// TwinCAT 3 PLC project FunctionBlocks
// ProgramVersion: 3.1.4023.0
// libraries:
//   Tc2_ControllerToolbox, * (Beckhoff Automation GmbH)
//   Tc2_Standard, * (Beckhoff Automation GmbH)
//   Tc2_System, * (Beckhoff Automation GmbH)
//   Tc3_Module, * (Beckhoff Automation GmbH)
// project tree:
//   DUTs/ dut_Auto_rock.TcDUT, dut_Brake.TcDUT, dut_Clutch.TcDUT, dut_Dol_Starter.TcDUT, ST_CSV_Record.TcDUT (not stored), S_Drive_control_settings.TcDUT, dut_hmi_Analogue.TcDUT, dut_hmi_Depth.TcDUT, dut_hmi_Drive_control.TcDUT, dut_hmi_Power_lever.TcDUT, dut_Least_gate.TcDUT, dut_Mode.TcDUT, dut_Power_lever.TcDUT, dut_Safety.TcDUT, S_TPD32_base_settings.TcDUT, S_General_settings.TcDUT
//   GVLs/ Brakes.TcGVL, Clutch.TcGVL, GVL.TcGVL, Mode.TcGVL, Power_lever.TcGVL, Safety.TcGVL, sp.TcGVL, Torque_prediction.TcGVL
//   / PlcTask.TcTTO
//   POUs/FBs/ FB_Brake_oil_pump.TcPOU, FB_Ctl_cmd_u.TcPOU, FB_DOL_Control.TcPOU, FB_Escort_monitoring.TcPOU, FB_Analogue.TcPOU, FB_Analogue_xcheck.TcPOU, FB_Auto_rock.TcPOU, FB_Backout.TcPOU, FB_BIT_TO_WORD_V0.TcPOU, FB_Brake.TcPOU, FB_Clutch.TcPOU, FB_Disc_brake.TcPOU, FB_Double_drum.TcPOU, FB_Drive_control.TcPOU, FB_Duty.TcPOU, FB_Encoder_depth.TcPOU, FB_Fast_brake.TcPOU, FB_Hysteresis.TcPOU, FB_Lag_filter.TcPOU, FB_Least_gate_element.TcPOU, FB_Least_gate_result.TcPOU, FB_Lincon.TcPOU, FB_Mode.TcPOU, FB_Motor_run_time.TcPOU, FB_Moving_average.TcPOU, FB_No_start.TcPOU, FB_Power_lever.TcPOU, FB_Raw_to_scaled.TcPOU, FB_Ref_ramp.TcPOU, FB_sp_write.TcPOU (not stored), FB_Standard_stuff.TcPOU, FB_Torque_prediction.TcPOU, FB_Torque_prediction_ST.TcPOU, FB_TPD_CANopen.TcPOU, FB_TP_with_stop.TcPOU, FB_Trip_control.TcPOU, FB_Valve_monitor.TcPOU, FB_Window.TcPOU, FB_WORD_TO_BIT_V0.TcPOU
//   POUs/ MAIN.TcPOU
//   POUs/Sections/ Winder_data.TcPOU
// real-time tasks:
//   TASK PlcTask: cycle T#10ms, priority 20, ADS port 350

CONFIGURATION FunctionBlocks
    RESOURCE PLC ON TwinCAT3
        TASK PlcTask(INTERVAL := T#10ms, PRIORITY := 20);
        PROGRAM MAIN WITH PlcTask : MAIN;
    END_RESOURCE
END_CONFIGURATION

// ---- DUTs/dut_Auto_rock.TcDUT
TYPE dut_Auto_rock :
STRUCT
	Status:WORD;
	Command:WORD;
END_STRUCT
END_TYPE

// ---- DUTs/dut_Brake.TcDUT
TYPE dut_Brake :
STRUCT
	Lh_off:BOOL;(*Left brake off signal - usually from left spring nest*)
	Lh_rubbing:BOOL; (*Left brake rubbing signal - usually from left spring nest*)
	Lh_on:BOOL; (*Left brake on signal - usually from left spring nest*)
	Lh_wear:BOOL; (*Left brake wear signal - usually from left spring nest*)
	Rh_off:BOOL; (*Right brake on signal - usually from right spring nest*)
	Rh_rubbing:BOOL; (*Right brake rubbing signal - usually from right spring nest*)
	Rh_on:BOOL; (*Right brake on signal - usually from right spring nest*)
	Rh_wear:BOOL; (*Right brake wear signal - usually from Right spring nest*)
	Lever_on:BOOL; (*Brake lever on limit switch*)
	Lever_off:BOOL; (*Brake lever off - normally from same limit switch as 'Lever_on'*)
	Lever_fully_off:BOOL; (*Brake lever fully off limit switch. Necessary for automatic winders.*)
	Maintenance_switch:BOOL; (*Brake maintenance switch (can be on driver's desk or in control panels).*)
	Maintenance_mode:BOOL;
	Lh_test:BOOL; (*Left brake test switch - normally on driver's desk. Often the same switch as Lh_dump.*)
	Rh_test:BOOL; (*Right brake test switch - normally on driver's desk. Often the same switch as Rh_dump.*)
	Lh_dump:BOOL; (*Left brake dump switch - normally on driver's desk. Often the same switch as Lh_test.*)
	Rh_dump:BOOL; (*Right brake dump switch - normally on driver's desk. Often the same switch as Rh_test.*)
	Proved_on:BOOL;
	Proved_on_500ms:BOOL;
END_STRUCT
END_TYPE

// ---- DUTs/dut_Clutch.TcDUT
TYPE dut_Clutch :
STRUCT
	Lh_in:BOOL;
	Lh_out:BOOL;
	Rh_in:BOOL;
	Rh_out:BOOL;
	Single_drum:BOOL;
END_STRUCT
END_TYPE

// ---- DUTs/dut_Dol_Starter.TcDUT
TYPE dut_Dol_Starter :
STRUCT
	Input_word:WORD; (*0=Switch, 1=Run, 2=Trip, 3=NoStart, 4=Estop, 5=IL1, 6=IL2, 7=IL3*)
	Output_word:WORD;
	Hrs:REAL;
	Minutes:REAL;
	Sec:REAL;
END_STRUCT
END_TYPE

// ---- DUTs/S_Drive_control_settings.TcDUT
TYPE S_Drive_control_settings :
STRUCT
	Max_drive_speed:INT;
	Max_drive_torque:INT;
	Speed_S_func_scans:INT;
	Current_S_func_scans:INT;
	No_start_time:TIME;
	Motor_fed_delay:TIME;
	Stall_time:TIME;
	Stall_speed:INT;
	Torque_ctrl_max_speed:INT;
	Brake_apply_speed:INT;
	Trail_brake_speed:INT;
	De_energise_to_trail:BOOL;
	Single_lever_control:BOOL;
	Stall_current:INT;
	Backout_min_speed:INT;

	(*Torque prediction settings*)	
	Lh_cage_mass_current:REAL;
	Rh_cage_mass_current:REAL;
	Lh_rope_mass_current:REAL;
	Rh_rope_mass_current:REAL;
	Full_payload_current:REAL;
	A_s2_per_m:REAL;
	Accel_torque_lag:TIME;
	Dynamic_friction_current:REAL;

END_STRUCT
END_TYPE

// ---- DUTs/dut_hmi_Analogue.TcDUT
TYPE dut_hmi_Analogue :
STRUCT
	Value:REAL;
	Per_thousand:REAL;
	Colour:INT;
END_STRUCT
END_TYPE

// ---- DUTs/dut_hmi_Depth.TcDUT
TYPE dut_hmi_Depth :
STRUCT
	Raw_count:REAL;
	Corrected_count:REAL;
	Raw_depth:REAL;
	Calibrated_depth:REAL;
	Compensated_depth:REAL;
	Offset:REAL;
	Speed:REAL;
	Status:WORD;
END_STRUCT
END_TYPE

// ---- DUTs/dut_hmi_Drive_control.TcDUT
TYPE dut_hmi_Drive_control :
STRUCT
	Speed_ref:INT;
	Torque_ref:INT;
	Torque_prediction:INT;
	Speed_scale:INT;
	Driver_ref_final:INT;
	Status:WORD;
END_STRUCT
END_TYPE

// ---- DUTs/dut_hmi_Power_lever.TcDUT
TYPE dut_hmi_Power_lever :
STRUCT
	Status:WORD;
	Raw:INT;
	Linear:INT;
	Cubic:INT;
END_STRUCT
END_TYPE

// ---- DUTs/dut_Least_gate.TcDUT
TYPE dut_Least_gate :
STRUCT
	Min_allowed_speed:REAL;
	Description:STRING[16];
	Rope_cap_mode:BOOL;
END_STRUCT
END_TYPE

// ---- DUTs/dut_Mode.TcDUT
TYPE dut_Mode :
STRUCT
	Manual:BOOL;
	Auto:BOOL;
	Auto_go:BOOL;
	Men:BOOL;
	Material:BOOL;
	Rope_capping:BOOL;
	Brake_maintenance:BOOL;
	Manual_switch:BOOL;
	Auto_switch:BOOL;
	Men_switch:BOOL;
	Material_switch:BOOL;
	Rope_capping_switch:BOOL;
	Rock:BOOL;
	Single_lever_control:BOOL;
END_STRUCT
END_TYPE

// ---- DUTs/dut_Power_lever.TcDUT
TYPE dut_Power_lever :
STRUCT
	Neutral:BOOL;
	Forward:BOOL;
	Reverse:BOOL;
	Button:BOOL;
	Raw:INT;
	Linear:INT;
	Cubic:INT;
END_STRUCT
END_TYPE

// ---- DUTs/dut_Safety.TcDUT
TYPE dut_Safety :
STRUCT
	Sc1:BOOL;
	Sc2:BOOL;
	Busc1:BOOL;
	Busc2:BOOL;
	Backup_safety_trip:BOOL;
	Main_safety_trip:BOOL;
	Lily_func_trip:BOOL;
	Lily_app_fault:BOOL;
	Backup_control_trip:BOOL;
	Control_trip:BOOL;
	Control_stop:BOOL;
	Lockout:BOOL;
	Enforced_slow:BOOL;
	Alarm:BOOL;
	All_clear:BOOL;
	Reset_button:BOOL;
	Reset_interlocks:BOOL;
	Reset:BOOL;
	Safe_for_power:BOOL;
	Bridge_present:BOOL;
END_STRUCT
END_TYPE

// ---- DUTs/S_TPD32_base_settings.TcDUT
TYPE S_TPD32_base_settings :
STRUCT
	Motor_base_rpm:REAL; (*Rated rpm of the motor*)
	Max_output_voltage:REAL; (*Maximum DC armature voltage*)
	Full_load_curr:REAL; (*Rated armature amps of the motor*)
	DCV_nominal_flux_current:REAL; (*Nominal flux current of the DCV according to S14 DIP switches*)
	Motor_nominal_flux_current:REAL; (*Nominal flux current of the DCV according to S14 DIP switches*)
	Flux_current_min:REAL; (*Percentage of rated motor field current for field weakening*)
	Acc_delta_time:REAL; (*Acceleration time from zero to rated motor rpm in seconds*)
	Dec_delta_time:REAL; (*Deceleration time from rated motor rpm to zero in seconds*)
END_STRUCT
END_TYPE

// ---- DUTs/S_General_settings.TcDUT
TYPE S_General_settings :
STRUCT
	Full_speed: REAL;
	Slow_switch_speed: REAL;
END_STRUCT
END_TYPE

// ---- GVLs/Brakes.TcGVL
{attribute 'qualified_only'}
VAR_GLOBAL
	Lh_off:BOOL;(*Left brake off signal - usually from left spring nest*)
	Lh_rubbing:BOOL; (*Left brake rubbing signal - usually from left spring nest*)
	Lh_on:BOOL; (*Left brake on signal - usually from left spring nest*)
	Lh_wear:BOOL; (*Left brake wear signal - usually from left spring nest*)
	Rh_off:BOOL; (*Right brake on signal - usually from right spring nest*)
	Rh_rubbing:BOOL; (*Right brake rubbing signal - usually from right spring nest*)
	Rh_on:BOOL; (*Right brake on signal - usually from right spring nest*)
	Rh_wear:BOOL; (*Right brake wear signal - usually from Right spring nest*)
	Lever_on:BOOL; (*Brake lever on limit switch*)
	Lever_off:BOOL; (*Brake lever off - normally from same limit switch as "Lever_on"*)
	Lever_fully_off:BOOL; (*Brake lever fully off limit switch. Necessary for automatic winders.*)
	Maintenance_switch:BOOL; (*Brake maintenance switch (can be on driver's desk or in control panels).*)
	Maintenance_mode:BOOL;
	Lh_test:BOOL; (*Left brake test switch - normally on driver's desk. Often the same switch as Lh_dump.*)
	Rh_test:BOOL; (*Right brake test switch - normally on driver's desk. Often the same switch as Rh_dump.*)
	Lh_dump:BOOL; (*Left brake dump switch - normally on driver's desk. Often the same switch as Lh_test.*)
	Rh_dump:BOOL; (*Right brake dump switch - normally on driver's desk. Often the same switch as Rh_test.*)
	Proved_on:BOOL;
	Proved_on_500ms:BOOL;
END_VAR

// ---- GVLs/Clutch.TcGVL
{attribute 'qualified_only'}
VAR_GLOBAL
	Lh_in:BOOL;
	Lh_out:BOOL;
	Rh_in:BOOL;
	Rh_out:BOOL;
	Single_drum:BOOL;
END_VAR

// ---- GVLs/GVL.TcGVL
{attribute 'qualified_only'}
VAR_GLOBAL
	Mode:dut_Mode;
	Brakes:dut_Brake;
	Clutch:dut_Clutch;
	Power_lever:dut_Power_lever;
	Safety:dut_Safety;
END_VAR

// ---- GVLs/Mode.TcGVL
{attribute 'qualified_only'}
VAR_GLOBAL
	Manual:BOOL;
	Auto:BOOL;
	Auto_go:BOOL;
	Men:BOOL;
	Material:BOOL;
	Rope_capping:BOOL;
	Brake_maintenance:BOOL;
	Manual_switch:BOOL;
	Auto_switch:BOOL;
	Men_switch:BOOL;
	Material_switch:BOOL;
	Rope_capping_switch:BOOL;
	Rock:BOOL;
	Single_lever_control:BOOL;
END_VAR

// ---- GVLs/Power_lever.TcGVL
{attribute 'qualified_only'}
VAR_GLOBAL
	Neutral:BOOL;
	Forward:BOOL;
	Reverse:BOOL;
	Button:BOOL;
	Raw:INT;
	Linear:INT;
	Cubic:INT;
END_VAR

// ---- GVLs/Safety.TcGVL
{attribute 'qualified_only'}
VAR_GLOBAL
	Sc1:BOOL;
	Sc2:BOOL;
	Busc1:BOOL;
	Busc2:BOOL;
	Backup_safety_trip:BOOL;
	Main_safety_trip:BOOL;
	Lily_func_trip:BOOL;
	Lily_app_fault:BOOL;
	Backup_control_trip:BOOL;
	Control_trip:BOOL;
	Control_stop:BOOL;
	Lockout:BOOL;
	Enforced_slow:BOOL;
	Alarm:BOOL;
	All_clear:BOOL;
	Reset_button:BOOL;
	Reset_interlocks:BOOL;
	Reset:BOOL;
	Safe_for_power:BOOL;
	Bridge_present:BOOL;
END_VAR

// ---- GVLs/sp.TcGVL
{attribute 'qualified_only'}
VAR_GLOBAL
	Gen: S_General_settings;
	Drive: S_Drive_control_settings;
	TPD: S_TPD32_base_settings;
END_VAR

// ---- GVLs/Torque_prediction.TcGVL
{attribute 'qualified_only'}
VAR_GLOBAL
	Lh_full: BOOL;
	Lh_half: BOOL;
	Equal: BOOL;
	Rh_half: BOOL;
	Rh_full: BOOL;
	
	Lh_full_request: BOOL;
	Lh_half_request: BOOL;
	Equal_request: BOOL;
	Rh_half_request: BOOL;
	Rh_full_request: BOOL;
END_VAR

// ---- POUs/MAIN.TcPOU
PROGRAM MAIN
VAR
END_VAR

END_PROGRAM

// ---- POUs/FBs/FB_Brake_oil_pump.TcPOU
FUNCTION_BLOCK FB_Brake_oil_pump
VAR_INPUT
	Run_cmd:BOOL;
	Stop_cmd:BOOL;
	Bop1_switch:BOOL;
	Bop1_tripped:BOOL;
	Bop1_running:BOOL;
	Bop1_use_internal_es:BOOL;
	Bop1_ext_estop:BOOL;
	Bop2_switch:BOOL;
	Bop2_tripped:BOOL;
	Bop2_running:BOOL;
	Bop2_use_internal_es:BOOL;
	Bop2_ext_estop:BOOL;
	Bop1_interlock:BOOL;
	Bop2_interlock:BOOL;
	Common_interlock:BOOL;
	Bridge1:BOOL;
	Bridge2:BOOL;
	Bridge3:BOOL;
	Pause_time:TIME;
	Reset:BOOL;
	Duty_bop1:REAL;
	Duty_bop2:REAL;
	Bop1_Reg455:REAL;
	Bop2_Reg455:REAL;
END_VAR
VAR_OUTPUT
	Bop1_run:BOOL;
	Bop2_run:BOOL;
	Bop1_ns_trip:BOOL;
	Bop1_es_trip:BOOL;
	Bop1_contactor_stuck:BOOL;
	Bop2_ns_trip:BOOL;
	Bop2_es_trip:BOOL;
	Bop2_contactor_stuck:BOOL;
	Start_output:BOOL;
	Bop1_Reg704:REAL;
	Bop1_Reg703:REAL;
	Bop1_Avg_curr:REAL;
	Bop2_Reg704:REAL;
	Bop2_Reg703:REAL;
	Bop2_Avg_curr:REAL;
END_VAR
VAR_IN_OUT
	Bop1_data:dut_Dol_Starter;
	Bop2_data:dut_Dol_Starter;
END_VAR
VAR
	FB_Duty_0: FB_Duty;
	FB_DOL_Control_0: FB_DOL_Control;
	FB_DOL_Control_1: FB_DOL_Control;
END_VAR

M_Brake_oil_pump();

METHOD M_Brake_oil_pump
VAR_INPUT
END_VAR
VAR_INST // added by the converter: edge detectors and wires of the graphical bodies
    _w1 : BOOL;
END_VAR
Start_output := _w1;
Bop1_avg_curr := FB_DOL_Control_0.Avg_curr;
Bop2_run := FB_DOL_Control_1.Fwd_command;
Bop1_run := FB_DOL_Control_0.Fwd_command;
Bop2_ns_trip := FB_DOL_Control_1.Ns_trip;
Bop2_es_trip := FB_DOL_Control_1.Estop_trip;
Bop2_contactor_stuck := FB_DOL_Control_1.Contactor_stuck;
Bop2_Reg704 := FB_DOL_Control_1.Reg_704;
Bop2_Reg703 := FB_DOL_Control_1.Reg_703;
_w1 := FB_DOL_Control_0.Start_output OR FB_DOL_Control_1.Start_output;
Bop1_ns_trip := FB_DOL_Control_0.Ns_trip;
Bop1_es_trip := FB_DOL_Control_0.Estop_trip;
Bop1_contactor_stuck := FB_DOL_Control_0.Contactor_stuck;
Bop1_Reg704 := FB_DOL_Control_0.Reg_704;
Bop2_avg_curr := FB_DOL_Control_1.Avg_curr;
Bop1_Reg703 := FB_DOL_Control_0.Reg_703;
FB_DOL_Control_1(
    Run_fwd := Run_cmd,
    Stop := Stop_cmd,
    Breaker_on := Bop2_switch,
    Breaker_tripped := Bop2_tripped,
    Contactor_feedback := Bop2_running,
    Interlock2 := Bop2_interlock,
    Bridge2 := Bridge2,
    Interlock3 := Common_interlock,
    Bridge3 := Bridge3,
    Reset := Reset,
    Use_internal_ES := Bop2_use_internal_es,
    Ext_estop := Bop2_ext_estop,
    Pause_time := Pause_time,
    Duty := FB_Duty_0.DutyB,
    Reg_455 := Bop2_Reg455,
    Starter_data := Bop2_data); // FB_DOL_Control
FB_DOL_Control_0(
    Run_fwd := Run_cmd,
    Stop := Stop_cmd,
    Breaker_on := Bop1_switch,
    Breaker_tripped := Bop1_tripped,
    Contactor_feedback := Bop1_running,
    Interlock1 := Bop1_interlock,
    Bridge1 := Bridge1,
    Interlock3 := Common_interlock,
    Bridge3 := Bridge3,
    Reset := Reset,
    Use_internal_ES := Bop1_use_internal_es,
    Ext_estop := Bop1_ext_estop,
    Pause_time := Pause_time,
    Duty := FB_Duty_0.DutyA,
    Reg_455 := Bop1_Reg455,
    Starter_data := Bop1_data); // FB_DOL_Control
FB_Duty_0(
    DutyA_times := Duty_bop1,
    DeviceA_running := Bop1_data.Input_word.1,
    DeviceA_switch := Bop1_data.Input_word.0,
    Force_dutyA := Bop1_data.Input_word.5,
    DutyB_times := Duty_bop2,
    Device_B_running := Bop2_data.Input_word.1,
    DeviceB_switch := Bop2_data.Input_word.0,
    Force_dutyB := Bop2_data.Input_word.5); // FB_Duty
END_METHOD

END_FUNCTION_BLOCK

// ---- POUs/FBs/FB_Duty.TcPOU
FUNCTION_BLOCK FB_Duty
VAR_INPUT
	DutyA_times:REAL; (*Times that Device A must run*)
	DeviceA_running:BOOL; (*Device A contactor feedback(running signal)*)
	DeviceA_switch:BOOL;
	DeviceA_ns:BOOL; (*Device A No Start - Switch duty to B*)
	Force_dutyA:BOOL;
	DutyB_times:REAL; (*Time that Device B must run*)
	DeviceB_running:BOOL; (*Device B contactor feedback(running signal)*)
	DeviceB_switch:BOOL;
	DeviceB_ns:BOOL; (*Device B No Start - Switch duty to A*)
	Force_dutyB:BOOL;
END_VAR
VAR_OUTPUT
	DutyA:BOOL; (*Device A output*)
	DutyB:BOOL; (*Device B output*)
END_VAR
VAR
	DeviceA_runtime:REAL;
	DeviceA_running_GT_1s:BOOL;
	DA_runtime:TIME;
	DeviceB_runtime:REAL;
	DeviceB_running_GT_1s:BOOL;
	DB_runtime:TIME;
	FE_bit_A :BOOL;
	FE_bit_B :BOOL;
	F_TRIG_0: F_TRIG;
	F_TRIG_1: F_TRIG;
	TON_2 : TON;
	TON_3 : TON;
END_VAR

M_Duty();

METHOD M_Duty
VAR_INPUT
END_VAR
IF NOT DeviceA_switch THEN
	DeviceA_runtime :=0;
end_if;
 
if NOT DeviceB_switch then
	DeviceB_runtime :=0;
end_if;

if NOT Force_dutyA and NOT Force_dutyB then
	if DeviceA_switch then
		IF DeviceA_runtime < DutyA_times AND NOT DutyB THEN
			DutyA := True;
		END_IF;
		F_TRIG_0(CLK:= DeviceA_running_GT_1s, Q=> FE_bit_A);
		IF FE_bit_A THEN
			DeviceA_runtime := DeviceA_runtime +1;
		end_if;
		if DeviceA_runtime >= DutyA_times and NOT Force_dutyA then
			DutyA := False;
			DeviceA_runtime := 0;
		end_if;

	end_if;


	if DeviceB_switch then
		IF DeviceB_runtime < DutyB_times AND NOT DutyA THEN
			DutyB := True;
		END_IF;
		F_TRIG_1(CLK:= DeviceB_running_GT_1s, Q=> FE_bit_B);
		IF FE_bit_B THEN
			DeviceB_runtime := DeviceB_runtime +1;
		end_if;
		if DeviceB_runtime >= DutyB_times and NOT Force_dutyB then
			DutyB := False;
			DeviceB_runtime := 0;
		end_if;
	end_if;

end_if;

if (Force_dutyA and DeviceA_switch) or (DeviceA_switch and NOT DeviceB_switch)  then
	DutyA := True;
	DutyB := False;
	DeviceA_runtime := 0;
	DeviceB_runtime := 0;
end_if;

if Force_dutyB and DeviceB_switch  or (DeviceB_switch and NOT DeviceA_switch) then
	DutyB := True;
	DutyA := False;
	DeviceA_runtime := 0;
	DeviceB_runtime := 0;
END_IF;

TON_2 (IN := DeviceA_running,
       PT := t#2s,
       Q => DeviceA_running_GT_1s,
       ET => DA_runtime);

TON_3 (IN := DeviceB_running,
       PT := t#2s,
       Q => DeviceB_running_GT_1s,
       ET => DB_runtime);
END_METHOD

END_FUNCTION_BLOCK

// ---- POUs/FBs/FB_DOL_Control.TcPOU
FUNCTION_BLOCK FB_DOL_Control
VAR_INPUT
	Run_fwd:BOOL; (*Pulsed Input to run forward*)
	Run_rev:BOOL; (*Pulsed Input to run reverse*)
	Stop:BOOL; (*Stop command*)
	Breaker_on:BOOL; (*Circuit breaker On status*)
	Breaker_tripped:BOOL;(*Overload tripped*)
	Contactor_feedback:BOOL; (*Running Feedback*)
	Interlock1:BOOL; (*Interlock to inhibit starter output*)
	Bridge1:BOOL; (*Bridge interlock1*)
	Interlock2:BOOL; (*Interlock to inhibit starter output*)
	Bridge2:BOOL; (*Bridge interlock2*)
	Interlock3:BOOL; (*Interlock to inhibit starter output*)
	Bridge3:BOOL; (*Bridge interlock3*)
	Reset:BOOL;
	Use_internal_ES:BOOL; (*1= Use EStop , 0= Dont use*)
	Ext_estop:BOOL; (*External Monitored Estop contact*)
	Pause_time:TIME; (*Time before starting next starter*)
	Duty:BOOL; (*1= active duty*)
	Hide_duty_indication:BOOL; (*1=Hide label on HMI*)
	Reg_455:REAL;
END_VAR
VAR_OUTPUT
	Fwd_command:BOOL; (*Run forward command*)
	Rev_command:BOOL; (*Run reverse command*)
	Ns_trip:BOOL;
	Estop_trip:BOOL; (*E-Stop/ Contactor feedback loss*)
	Contactor_stuck:BOOL; (*No run command but contactor closed*)
	Tripped_out:BOOL;
	Start_output:BOOL; (*Start command to next starter block*)
	Reg_704:REAL;
	Reg_703:REAL;
	Avg_curr:REAL;
END_VAR
VAR_IN_OUT
	Starter_data:dut_Dol_Starter;
END_VAR
VAR
	No_start:BOOL;
	Estop:BOOL;
	Invalid_cmd:BOOL;
	Motor_hrs:REAL;
	Motor_min:REAL;
	Motor_sec:REAL;
	hmi_Run_fwd:BOOL;
	hmi_Run_rev:BOOL;
	hmi_Stop:BOOL;
	hmi_Manual:BOOL;
	hmi_Rst_run_time:BOOL;
	hmi_Force_duty:BOOL;
	CAN_cb_on:BOOL;
	CAN_tripped:BOOL;
	CAN_running:BOOL;
	Cb_on:BOOL;
	Running:BOOL;
	Tripped:BOOL;
	Q:BOOL;
	FB_BIT_TO_WORD_V0_0: FB_BIT_TO_WORD_V0;
	FB_WORD_TO_BIT_V0_0: FB_WORD_TO_BIT_V0;
	FB_Ctl_cmd_u_0: FB_Ctl_cmd_u;
	RS_0: RS;
	TON_0: TON;
	RS_1: RS;
	RS_2: RS;
	FB_No_start_0: FB_No_start;
	FB_Motor_run_time_0: FB_Motor_run_time;
	TOF_0: TOF;
	F_TRIG_0: F_TRIG;
	R_TRIG_0: R_TRIG;
	RS_3: RS;
	TON_1: TON;
	R_TRIG_1: R_TRIG;
	R_TRIG_2: R_TRIG;
END_VAR

M_Pack_data();
M_Starter_control();
M_No_start();
M_Motor_run_time();
M_Cascade_function();

METHOD M_Cascade_function
VAR_INPUT
END_VAR
VAR_INST // added by the converter: edge detectors and wires of the graphical bodies
    _w1, _w2, _w4 : BOOL;
    _w3 : ANY;
END_VAR
_w2 := F_TRIG_0.Q OR _w1 OR R_TRIG_1.Q AND No_start;
F_TRIG_0(CLK := TOF_0.Q); // F_TRIG
R_TRIG_2(CLK := _w3); // R_TRIG
_w4 := Run_fwd OR Run_rev;
TOF_0(IN := 1 AND _w4 AND NOT hmi_Manual, PT := Pause_time); // TOF
Start_output := R_TRIG_2.Q;
_w1 := _w4 AND hmi_Manual;
R_TRIG_0(CLK := _w4); // R_TRIG
RS_3(SET := R_TRIG_0.Q); // RS
Q := RS_3.Q1;
TON_1(IN := Q, PT := t#2s); // TON
(* Stop OR TON_1.Q; result not used *)
R_TRIG_1(CLK := TON_1.Q); // R_TRIG
_w3 := _w2 AND Duty;
END_METHOD

METHOD M_Motor_run_time
VAR_INPUT
END_VAR
Motor_hrs := FB_Motor_run_time_0.Hours;
Motor_min := FB_Motor_run_time_0.Minutes;
Motor_sec := FB_Motor_run_time_0.Sec;
FB_Motor_run_time_0(Start := Running, Reset := hmi_Rst_run_time); // FB_Motor_run_time
END_METHOD

METHOD M_No_start
VAR_INPUT
END_VAR
VAR_INST // added by the converter: edge detectors and wires of the graphical bodies
    _w1 : BOOL;
END_VAR
No_start := FB_No_start_0.NS_trip;
Estop := FB_No_start_0.Estop_out;
Ns_trip := _w1;
Estop_trip := Estop;
FB_No_start_0(
    Run := Fwd_command OR Rev_command,
    No_start_trip := No_start,
    Reset := Reset,
    Run_FB := Running,
    CB_trip := Tripped,
    CB_On := Cb_on,
    Use_int_estop := Use_internal_ES,
    Ext_estop := Ext_estop,
    Ns_time := t#5s); // FB_No_start
_w1 := No_start;
END_METHOD

METHOD M_Pack_data
VAR_INPUT
END_VAR
Tripped_out := Tripped;
Running := Contactor_feedback OR CAN_running;
CB_on := Breaker_on OR CAN_cb_on;
Tripped := CAN_tripped OR Breaker_tripped;
hmi_Run_rev := FB_WORD_TO_BIT_V0_0.bit1;
hmi_Stop := FB_WORD_TO_BIT_V0_0.bit2;
hmi_Manual := FB_WORD_TO_BIT_V0_0.bit3;
hmi_Rst_run_time := FB_WORD_TO_BIT_V0_0.bit4;
hmi_Force_duty := FB_WORD_TO_BIT_V0_0.bit5;
FB_WORD_TO_BIT_V0_0(Word_in := Starter_data.Output_word); // FB_WORD_TO_BIT_V0
hmi_Run_fwd := FB_WORD_TO_BIT_V0_0.bit0;
// Bits to HMI for indication
FB_BIT_TO_WORD_V0_0(
    bit0 := CB_on,
    bit1 := Running,
    bit2 := Tripped,
    bit3 := No_start,
    bit4 := Estop,
    bit5 := Interlock1,
    bit6 := Interlock2,
    bit7 := Interlock3,
    bit8 := Duty,
    bit9 := Hide_duty_indication); // FB_BIT_TO_WORD_V0
Starter_data.Input_word := FB_BIT_TO_WORD_V0_0.Word_out;
Reg_704 := FB_Ctl_cmd_u_0.Reg_704;
Reg_703 := FB_Ctl_cmd_u_0.Reg_703;
CAN_cb_on := FB_Ctl_cmd_u_0.Ready;
CAN_tripped := FB_Ctl_cmd_u_0.Tripped;
CAN_running := FB_Ctl_cmd_u_0.Running;
Avg_curr := FB_Ctl_cmd_u_0.Avg_curr;
Starter_data.Minutes := Motor_min;
Starter_data.Sec := Motor_sec;
// Input_word.0 -> Switch
// Input_word.1 -> Running
// Input_word.2 -> Trip
// Input_word.3 -> No Start
// Input_word.4 -> EStop
// Input_word.5 -> Interlock 1
// Input_word.6 -> Interlock 2
// Input_word.7 -> Interlock 3
// Output_word.0 -> Run Fwd
// Output_word.1 -> Run Rev
// Output_word.2 -> Stop
// Output_word.3 -> Auto = 0,
// Manual = 1
//
Starter_data.Hrs := Motor_hrs;
FB_Ctl_cmd_u_0(
    Reg_455 := REAL_TO_INT(Reg_455),
    Run_fwd := Fwd_command,
    Run_rev := Rev_command,
    Rst_flt := Reset,
    Rst_warn := Reset); // FB_Ctl_cmd_u
END_METHOD

METHOD M_Starter_control
VAR_INPUT
END_VAR
VAR_INST // added by the converter: edge detectors and wires of the graphical bodies
    _w1, _w2, _w4, _w5, _w6, _w7, _w8, _w9, _w10 : BOOL;
    _w3, _w11 : ANY;
END_VAR
RS_0(SET := _w1 OR _w2, RESET1 := _w3); // RS
Invalid_cmd := _w4;
// Forward command
_w1 := hmi_Manual AND hmi_Run_fwd;
_w2 := NOT hmi_Manual AND Run_fwd;
Rev_command := RS_1.Q1;
_w5 := Bridge1 AND hmi_Manual;
_w3 := Interlock1 AND NOT (Bridge1 AND hmi_Manual) OR Interlock2 AND NOT (Bridge1 AND hmi_Manual) OR _w6 OR No_start OR Estop OR NOT Cb_on OR Stop OR Invalid_cmd OR _w7 OR NOT Duty OR Tripped;
_w7 := hmi_Stop AND Running;
_w4 := Run_fwd AND Run_rev;
Fwd_command := RS_0.Q1;
Contactor_stuck := RS_2.Q1;
// Reverse command
RS_1(SET := hmi_Manual AND hmi_Run_rev OR _w10, RESET1 := Interlock1 AND NOT Bridge1 AND NOT hmi_Manual OR Interlock2 AND NOT Bridge2 AND NOT hmi_Manual OR _w8 OR No_start OR Estop OR NOT Breaker_on OR Stop OR Invalid_cmd OR _w9 OR NOT Duty); // RS
_w10 := NOT hmi_Manual AND Run_rev;
_w6 := Interlock3 AND NOT _w5;
_w8 := Interlock3 AND NOT Bridge3 AND NOT hmi_Manual;
TON_0(IN := _w11, PT := t#500ms); // TON
_w11 := NOT Fwd_command AND Contactor_feedback AND NOT Rev_command;
_w9 := hmi_Stop AND Contactor_feedback;
// CAN portion not done for reverse
RS_2(SET := TON_0.Q, RESET1 := Reset); // RS
END_METHOD

END_FUNCTION_BLOCK

// ---- POUs/FBs/FB_BIT_TO_WORD_V0.TcPOU
FUNCTION_BLOCK FB_BIT_TO_WORD_V0
VAR_INPUT
	bit0:BIT;
	bit1:BIT;
	bit2:BIT;
	bit3:BIT;
	bit4:BIT;
	bit5:BIT;
	bit6:BIT;
	bit7:BIT;
	bit8:BIT;
	bit9:BIT;
	bit10:BIT;
	bit11:BIT;
	bit12:BIT;
	bit13:BIT;
	bit14:BIT;
	bit15:BIT;
END_VAR
VAR_OUTPUT
	Word_out:WORD;
END_VAR
VAR
END_VAR
VAR // added by the converter: edge detectors and wires of the graphical bodies
    _w1, _w2, _w3, _w4, _w5, _w6, _w7, _w8, _w9, _w10, _w11, _w12, _w13, _w14, _w15 : ANY;
END_VAR

Word_out.1 := _w1;
Word_out.9 := _w2;
Word_out.2 := _w3;
Word_out.10 := _w4;
Word_out.3 := _w5;
Word_out.11 := _w6;
Word_out.4 := _w7;
Word_out.12 := _w8;
Word_out.5 := _w9;
Word_out.13 := _w10;
Word_out.6 := _w11;
Word_out.14 := _w12;
Word_out.7 := _w13;
Word_out.15 := _w14;
Word_out.8 := _w15;
// Pack bits into a word
_w1 := bit1;
_w2 := bit9;
_w3 := bit2;
_w4 := bit10;
_w5 := bit3;
_w6 := bit11;
_w7 := bit4;
_w8 := bit12;
_w9 := bit5;
_w10 := bit13;
_w11 := bit6;
_w12 := bit14;
_w13 := bit7;
_w14 := bit15;
_w15 := bit8;
Word_out.0 := bit0;

END_FUNCTION_BLOCK

// ---- POUs/FBs/FB_WORD_TO_BIT_V0.TcPOU
FUNCTION_BLOCK FB_WORD_TO_BIT_V0
VAR_INPUT
	Word_in:WORD;
END_VAR
VAR_OUTPUT
	bit0:BIT;
	bit1:BIT;
	bit2:BIT;
	bit3:BIT;
	bit4:BIT;
	bit5:BIT;
	bit6:BIT;
	bit7:BIT;
	bit8:BIT;
	bit9:BIT;
	bit10:BIT;
	bit11:BIT;
	bit12:BIT;
	bit13:BIT;
	bit14:BIT;
	bit15:BIT;
END_VAR
VAR
END_VAR

// Unpacks a word into bits
bit0 := Word_in.0;
bit8 := Word_in.8;
bit1 := Word_in.1;
bit9 := Word_in.9;
bit2 := Word_in.2;
bit10 := Word_in.10;
bit3 := Word_in.3;
bit11 := Word_in.11;
bit4 := Word_in.4;
bit12 := Word_in.12;
bit5 := Word_in.5;
bit13 := Word_in.13;
bit6 := Word_in.6;
bit14 := Word_in.14;
bit7 := Word_in.7;
bit15 := Word_in.15;

END_FUNCTION_BLOCK

// ---- POUs/FBs/FB_Ctl_cmd_u.TcPOU
FUNCTION_BLOCK FB_Ctl_cmd_u
VAR_INPUT
	Reg_455:INT;
	Run_fwd:BOOL;
	Run_rev:BOOL;
	Rst_flt:BOOL;
	Rst_warn:BOOL;
	Ther_ov_test:BOOL;
	Trip_tst:BOOL;
END_VAR
VAR_OUTPUT
	Reg_704:INT;
	Reg_703:INT;
	Ready:BOOL;
	Closed:BOOL;
	Tripped:BOOL;
	Fault:BOOL;
	Alarm:BOOL;
	Rst_auth:BOOL;
	Starting:BOOL;
	Running:BOOL;
	Avg_curr:REAL;
END_VAR
VAR
END_VAR
{warning 'TODO: This needs to be replicated for our equiment'}

(* Command treatment *)
IF Run_fwd THEN Run_fwd S= Reg_704.0;
ELSE Run_fwd R= Reg_704.0;
END_IF;
     
IF Run_rev THEN Run_rev S= Reg_704.1;
ELSE Run_rev R= Reg_704.1;
END_IF;
     
IF Rst_flt THEN Rst_flt S=Reg_704.3;
ELSE Rst_flt R= Reg_704.3;
END_IF;
     
IF Ther_ov_test THEN Ther_ov_test S= Reg_704.5;
ELSE Ther_ov_test R= Reg_704.5;
END_IF;
     
IF Trip_tst THEN Trip_tst S= Reg_704.12;
ELSE Trip_tst R= Reg_704.12;
END_IF;

IF Rst_warn THEN Rst_warn S= Reg_703.3;
ELSE Rst_warn R= Reg_703.3;
END_IF;

(* Controltreatment *)
Ready := Reg_455.0;
Closed := Reg_455.1;
Fault := Reg_455.2;
Alarm := Reg_455.3;
Tripped := Reg_455.4;
Rst_auth := Reg_455.5;
Running := Reg_455.7;
Starting := Reg_455.15;
Avg_curr := Reg_455 AND 16128;
Avg_curr := SHRZ_INT(Avg_curr,8);
Avg_curr := Avg_curr * 318 / 100;

END_FUNCTION_BLOCK

// ---- POUs/FBs/FB_No_start.TcPOU
FUNCTION_BLOCK FB_No_start
VAR_INPUT
	Run:BOOL;
	No_start_trip:BOOL;
	Reset:BOOL;
	Run_FB:BOOL;
	CB_trip:BOOL;
	CB_On:BOOL;
	Use_int_estop:BOOL; (*Internally generated E-Stop when Contactor feedback is lost without removing run command*)
	Ext_estop:BOOL; (*External Estop with monitored contact*)
	Ns_time:TIME;
END_VAR
VAR_OUTPUT
	NS_trip:BOOL;
	Estop_out:BOOL;
END_VAR
VAR
	TON_0: TON;
	SR_0: SR;
	F_TRIG_0: F_TRIG;
	SR_1: SR;
END_VAR

M_Main();

METHOD M_Main
VAR_INPUT
END_VAR
VAR_INST // added by the converter: edge detectors and wires of the graphical bodies
    _w1, _w3, _w4 : BOOL;
    _w2 : ANY;
END_VAR
Estop_out := SR_1.Q1;
Ns_trip := SR_0.Q1;
_w1 := (F_TRIG_0.Q AND Run AND NOT NS_trip AND NOT CB_trip) AND Use_int_estop;
SR_1(SET1 := _w2, RESET := Reset); // SR
_w4 := _w3 AND NOT Run_FB;
_w3 := Run AND NOT No_start_trip AND CB_On AND NOT Estop_out;
TON_0(IN := _w4, PT := Ns_time); // TON
SR_0(SET1 := TON_0.Q, RESET := Reset); // SR
F_TRIG_0(CLK := Run_FB); // F_TRIG
_w2 := Ext_estop OR _w1;
END_METHOD

END_FUNCTION_BLOCK

// ---- POUs/FBs/FB_Motor_run_time.TcPOU
FUNCTION_BLOCK FB_Motor_run_time
VAR_INPUT
	Start:BOOL;
	Reset:BOOL;
END_VAR
VAR_OUTPUT
	Hours:REAL;
	Minutes:REAL;
	Sec:REAL;
END_VAR
VAR
	T2_dn:BOOL;
	one_sec_pulse:BOOL;
	Min_pulse:BOOL;
	Hour_pulse:BOOL;
	End_pulse:BOOL;
	TON_0: TON;
	TON_1: TON;
	R_TRIG_0: R_TRIG;
	CTU_0: CTU;
	R_TRIG_1: R_TRIG;
	R_TRIG_2: R_TRIG;
	CTU_1: CTU;
	CTU_2: CTU;
END_VAR

M_Main();

METHOD M_Main
VAR_INPUT
END_VAR
VAR_INST // added by the converter: edge detectors and wires of the graphical bodies
    _w1, _w2 : ANY;
END_VAR
T2_dn := TON_1.Q;
Minutes := CTU_1.CV;
one_sec_pulse := R_TRIG_0.Q;
IF Start THEN
    TON_1(IN := NOT TON_0.Q, PT := t#500ms); // TON
END_IF
Hour_pulse := CTU_1.Q;
R_TRIG_0(CLK := TON_0.Q); // R_TRIG
Min_pulse := CTU_0.Q;
Sec := CTU_0.CV;
CTU_1(CU := R_TRIG_1.Q, RESET := Hour_pulse OR Reset, PV := 60); // CTU
IF Start THEN
    TON_0(IN := T2_dn, PT := t#500ms); // TON
END_IF
CTU_0(CU := one_sec_pulse, RESET := _w1, PV := 60); // CTU
// Seconds
_w1 := Min_pulse OR Reset;
// Minutes
R_TRIG_1(CLK := Min_pulse); // R_TRIG
// Hours
R_TRIG_2(CLK := Hour_pulse); // R_TRIG
CTU_2(CU := R_TRIG_2.Q, RESET := _w2, PV := 32767); // CTU
_w2 := End_pulse OR Reset;
End_pulse := CTU_2.Q;
Hours := CTU_2.CV;
END_METHOD

END_FUNCTION_BLOCK

// ---- POUs/FBs/FB_Escort_monitoring.TcPOU
FUNCTION_BLOCK FB_Escort_monitoring
VAR_INPUT
	Coil_Lh1:BOOL;
	Coil_Lh2:BOOL;
	Coil_Rh1:BOOL;
	Coil_Rh2:BOOL;
	Valve_Lh1_open:BOOL;
	Valve_Lh1_closed:BOOL;
	Valve_Lh2_open:BOOL;
	Valve_Lh2_closed:BOOL;
	Valve_Rh1_open:BOOL;
	Valve_Rh1_closed:BOOL;
	Valve_Rh2_open:BOOL;
	Valve_Rh2_closed:BOOL;
	Open_time:TIME;
	Close_time:TIME;
END_VAR
VAR_OUTPUT
	Lh1_not_opening:BOOL;
	Lh1_not_closing:BOOL;
	Lh1_open_and_closed:BOOL;
	Lh2_not_opening:BOOL;
	Lh2_not_closing:BOOL;
	Lh2_open_and_closed:BOOL;
	Rh1_not_opening:BOOL;
	Rh1_not_closing:BOOL;
	Rh1_open_and_closed:BOOL;
	Rh2_not_opening:BOOL;
	Rh2_not_closing:BOOL;
	Rh2_open_and_closed:BOOL;
	Lh1_with_brakes_on:BOOL;
	Lh2_with_brakes_on:BOOL;
	Rh1_with_brakes_on:BOOL;
	Rh2_with_brakes_on:BOOL;
	Lh1_Lh2_xcheck:BOOL;
	Rh1_Rh2_xcheck:BOOL;
	Lh1_chatter:BOOL;
	Lh2_chatter:BOOL;
	Rh1_chatter:BOOL;
	Rh2_chatter:BOOL;
END_VAR
VAR
	Reset_chatter_counters:BOOL;
	FB_Valve_monitor_0: FB_Valve_monitor;
	FB_Valve_monitor_1: FB_Valve_monitor;
	FB_Valve_monitor_2: FB_Valve_monitor;
	FB_Valve_monitor_3: FB_Valve_monitor;
	TON_0: TON;
	TON_1: TON;
	TON_2: TON;
	TON_3: TON;
	R_TRIG_0: R_TRIG;
	CTU_0: CTU;
	CTU_1: CTU;
	CTU_2: CTU;
	CTU_3: CTU;
END_VAR

M_Escort_valves();

METHOD M_Escort_valves
VAR_INPUT
END_VAR
{warning 'TODO: Address %S7 needs to be correctly addressed'}
VAR_INST // added by the converter: edge detectors and wires of the graphical bodies
    _w1, _w5 : ANY;
    _w2, _w3, _w4 : BOOL;
END_VAR
Rh2_not_opening := FB_Valve_monitor_3.Not_opening;
TON_3(IN := _w1, PT := t#100ms); // TON
Rh1_with_brakes_on := _w2;
Lh1_open_and_closed := FB_Valve_monitor_0.Open_and_closed;
Rh2_not_closing := FB_Valve_monitor_3.Not_closing;
Rh1_not_opening := FB_Valve_monitor_2.Not_opening;
Rh2_open_and_closed := FB_Valve_monitor_3.Open_and_closed;
Rh1_not_closing := FB_Valve_monitor_2.Not_closing;
_w3 := Coil_Rh2 AND TON_1.Q;
Rh1_open_and_closed := FB_Valve_monitor_2.Open_and_closed;
Lh2_open_and_closed := FB_Valve_monitor_1.Open_and_closed;
Lh1_not_closing := FB_Valve_monitor_0.Not_closing;
FB_Valve_monitor_3(
    Coil_state := Coil_Rh2,
    Energise_to_open := 0,
    Valve_open := Valve_Rh2_open,
    Valve_closed := Valve_Rh2_closed,
    Open_time := Open_time,
    Close_time := Close_time); // FB_Valve_monitor
Lh2_not_opening := FB_Valve_monitor_1.Not_opening;
Lh2_not_closing := FB_Valve_monitor_1.Not_closing;
Lh1_with_brakes_on := _w4;
Lh2_with_brakes_on := Coil_Lh2 AND TON_0.Q;
TON_2(IN := _w5, PT := t#100ms); // TON
_w1 := Coil_Rh1 XOR Coil_Rh2;
Rh1_Rh2_xcheck := TON_3.Q;
Lh1_Lh2_xcheck := TON_2.Q;
Lh1_chatter := CTU_0.Q;
CTU_1(CU := Coil_Rh1, RESET := Reset_chatter_counters, PV := 10); // CTU
_w2 := Coil_Rh1 AND TON_1.Q;
FB_Valve_monitor_2(
    Coil_state := Coil_Rh1,
    Energise_to_open := 0,
    Valve_open := Valve_Rh1_open,
    Valve_closed := Valve_Rh1_closed,
    Open_time := Open_time,
    Close_time := Close_time); // FB_Valve_monitor
Lh1_not_opening := FB_Valve_monitor_0.Not_opening;
Rh2_with_brakes_on := _w3;
FB_Valve_monitor_1(
    Coil_state := Coil_Lh2,
    Energise_to_open := 0,
    Valve_open := Valve_Lh2_open,
    Valve_closed := Valve_Lh2_closed,
    Open_time := Open_time,
    Close_time := Close_time); // FB_Valve_monitor
Rh1_chatter := CTU_1.Q;
TON_1(IN := Brakes.Rh_on, PT := t#10s); // TON
FB_Valve_monitor_0(
    Coil_state := Coil_Lh1,
    Energise_to_open := 0,
    Valve_open := Valve_Lh1_open,
    Valve_closed := Valve_Lh1_closed,
    Open_time := Open_time,
    Close_time := Close_time); // FB_Valve_monitor
_w4 := Coil_Lh1 AND TON_0.Q;
TON_0(IN := Brakes.Lh_on, PT := t#10s); // TON
_w5 := Coil_Lh1 XOR Coil_Lh2;
R_TRIG_0(CLK := %S7); // R_TRIG
Reset_chatter_counters := R_TRIG_0.Q OR NOT Safety.Sc1 OR Safety.Reset OR NOT Brakes.Lh_on OR NOT Brakes.Rh_on;
// This address needs to be changed
CTU_0(CU := Coil_Lh1, RESET := Reset_chatter_counters, PV := 10); // CTU
CTU_2(CU := Coil_Lh2, RESET := Reset_chatter_counters, PV := 10); // CTU
CTU_3(CU := Coil_Rh2, RESET := Reset_chatter_counters, PV := 10); // CTU
Lh2_chatter := CTU_2.Q;
Rh2_chatter := CTU_3.Q;
END_METHOD

END_FUNCTION_BLOCK

// ---- POUs/FBs/FB_Valve_monitor.TcPOU
FUNCTION_BLOCK FB_Valve_monitor
VAR_INPUT
	Coil_state:BOOL;
	Energise_to_open:BOOL;
	Valve_open:BOOL;
	Valve_closed:BOOL;
	Open_time:TIME;
	Close_time:TIME;
END_VAR
VAR_OUTPUT
	Not_opening:BOOL;
	Not_closing:BOOL;
	Open_and_closed:BOOL;
END_VAR
VAR
	TON_0: TON;
END_VAR

M_Valve_monitor();

METHOD M_Valve_monitor
VAR_INPUT
END_VAR
VAR_INST // added by the converter: edge detectors and wires of the graphical bodies
    _w1 : BOOL;
END_VAR
_w1 := Valve_open AND Valve_closed;
Not_closing := TON_0.Q;
Not_opening := TON_0.Q;
TON_0(IN := NOT (Coil_state XOR Energise_to_open) AND NOT Valve_closed, PT := Close_time); // TON
Open_and_closed := _w1;
TON_0(IN := NOT (Coil_state XOR Energise_to_open) AND NOT Valve_open, PT := Open_time); // TON
END_METHOD

END_FUNCTION_BLOCK

// ---- POUs/FBs/FB_Analogue.TcPOU
FUNCTION_BLOCK FB_Analogue
VAR_INPUT
	Value:REAL;
	Raw_min:REAL;
	Raw_max:REAL;
	Scaled_min:REAL;
	Scaled_max:REAL;
	HH_setpoint:REAL := 1.000000E+008; (*The default value prevents the output from triggering if no setpoint is given*)
	H_setpoint:REAL := 1.000000E+008;
	L_setpoint:REAL := -1.000000E+008;
	LL_setpoint:REAL := -1.000000E+008;
	Hysteresis:REAL;
	Filter_time:TIME;
	Alarm_inhibit_time:TIME;
	HMI_min:REAL;
	HMI_max:REAL;
	Colour_scheme:INT;
END_VAR
VAR_OUTPUT
	Scaled_value:REAL;
	HH:BOOL;
	H:BOOL;
	L:BOOL;
	LL:BOOL;
	HMI:dut_hmi_Analogue;
END_VAR
VAR
	TON_0: TON;
	TON_1: TON;
	TON_2: TON;
	TON_3: TON;
END_VAR

M_Analogue();
M_Analogue_HMI();

METHOD M_Analogue
VAR_INPUT
END_VAR
{warning "TODO: the LEAD LAG filter needs to be looked at by Bret so that he can make sure it does what he needs it to."}
{warning "TODO: the HYST FB needs to be looked at by Bret so that he can make sure it does what he needs it to."}
VAR
	LF0: FB_Lag_filter;
	FB_Hysteresis_0: FB_Hysteresis;
	FB_Hysteresis_1: FB_Hysteresis;
	FB_Hysteresis_2: FB_Hysteresis;
	FB_Hysteresis_3: FB_Hysteresis;
END_VAR
VAR_INST // added by the converter: edge detectors and wires of the graphical bodies
    _w1 : REAL;
END_VAR
FB_Hysteresis_1(In := Scaled_value, On_val := H_setpoint + Hysteresis, Off_val := H_setpoint); // FB_Hysteresis
TON_1(IN := FB_Hysteresis_1.Out, PT := Alarm_inhibit_time); // TON
H := TON_1.Q;
_w1 := LF0.Out - Raw_min;
// Convert integer value to real, then apply filtering and scaling
LF0(In := Value, Time_const := Filter_time); // FB_Lag_filter
Scaled_value := (_w1 / (Raw_max - Raw_min)) * (Scaled_max - Scaled_min) + Scaled_min;
TON_0(IN := FB_Hysteresis_0.Out, PT := Alarm_inhibit_time); // TON
// Alarms
FB_Hysteresis_0(In := Scaled_value, On_val := HH_setpoint + Hysteresis, Off_val := HH_setpoint); // FB_Hysteresis
HH := TON_0.Q;
FB_Hysteresis_2(In := Scaled_value, On_val := L_setpoint + Hysteresis, Off_val := L_setpoint); // FB_Hysteresis
TON_2(IN := NOT FB_Hysteresis_2.Out, PT := Alarm_inhibit_time); // TON
L := TON_2.Q;
FB_Hysteresis_3(In := Scaled_value, On_val := LL_setpoint + Hysteresis, Off_val := LL_setpoint); // FB_Hysteresis
TON_3(IN := NOT FB_Hysteresis_3.Out, PT := Alarm_inhibit_time); // TON
LL := TON_3.Q;
END_METHOD

METHOD M_Analogue_HMI
VAR_INPUT
END_VAR
VAR_INST // added by the converter: edge detectors and wires of the graphical bodies
    _w1, _w2, _w3, _w4, _w5, _w6, _w7 : ANY;
END_VAR
_w2 := LIMIT(-1000, _w1, 1000);
_w1 := _w3 * 1000;
IF Scaled_value >= HH_setpoint THEN _w4 := 0; END_IF
HMI.Colour := _w4;
// Pack HMI values into structure. First the scaled value (in correct units), then the percentage value - limited to 0% to 100%.
HMI.Value := Scaled_value;
_w3 := (Scaled_value - HMI_min) / (HMI_max - HMI_min);
HMI.Per_thousand := _w2;
HMI.Colour := 2;
IF Scaled_value >= H_setpoint THEN _w5 := 1; END_IF
HMI.Colour := _w5;
IF Scaled_value <= L_setpoint THEN _w6 := 3; END_IF
HMI.Colour := _w6;
IF Scaled_value <= LL_setpoint THEN _w7 := 4; END_IF
HMI.Colour := _w7;
HMI.Colour := (Colour_scheme - 1) * 5 + HMI.Colour;
END_METHOD

END_FUNCTION_BLOCK

// ---- POUs/FBs/FB_Lag_filter.TcPOU
FUNCTION_BLOCK FB_Lag_filter
VAR_INPUT
	In: REAL;
	Time_const: TIME;
END_VAR
VAR_OUTPUT
	Out: REAL;
END_VAR
VAR	
	fbGetCurTaskIdx  : GETCURTASKINDEX;
	Scan_time: REAL;
	T: REAL;
END_VAR

Scan_time:= UINT_TO_REAL(_TaskInfo[fbGetCurTaskIdx.index].CycleTime) / 10.0;
T:= TIME_TO_REAL(Time_const);

Out:= Out + (In - Out) * Scan_Time / (T - Scan_time);

END_FUNCTION_BLOCK

// ---- POUs/FBs/FB_Hysteresis.TcPOU
FUNCTION_BLOCK FB_Hysteresis
VAR_INPUT
	In: REAL;
	On_val: REAL;
	Off_val: REAL;
END_VAR
VAR_OUTPUT
	Out: BOOL;
END_VAR
VAR	
END_VAR

IF In > On_val THEN
	Out:= TRUE;
END_IF
IF In < Off_val THEN
	Out:= FALSE;
END_IF

END_FUNCTION_BLOCK

// ---- POUs/FBs/FB_Analogue_xcheck.TcPOU
FUNCTION_BLOCK FB_Analogue_xcheck
VAR_INPUT
	In1:REAL;
	In2:REAL;
	Constant_window:REAL;
	Percent_window:REAL;
	Use_absolute_values:BOOL;
END_VAR
VAR_OUTPUT
	Mismatch:BOOL;
END_VAR
VAR
END_VAR

M_Analogue_xcheck();

METHOD M_Analogue_xcheck
VAR_INPUT
END_VAR
VAR_INST // added by the converter: edge detectors and wires of the graphical bodies
    _w1, _w2, _w3 : ANY;
END_VAR
Mismatch := ABS(_w1 - _w2) > _w3;
_w2 := SEL(Use_absolute_values, In2, ABS(In2));
_w1 := SEL(Use_absolute_values, In1, ABS(In1));
_w3 := (Percent_window / 100) * (ABS(In1)) + Constant_window;
END_METHOD

END_FUNCTION_BLOCK

// ---- POUs/FBs/FB_Auto_rock.TcPOU
FUNCTION_BLOCK FB_Auto_rock
VAR_INPUT
	Safety_interlock:BOOL;
	Lh_depth:REAL;
	Rh_depth:REAL;
	Underground_despatch:BOOL;
	Right_brakes_on_dist:REAL;
	Left_brakes_on_dist:REAL;
	Tip_zone_up:REAL;
	Tip_zone_down:REAL;
	Box_zone_up:REAL;
	Box_zone_down:REAL;
	Rock_cycle_unlatch_dist:REAL;
	Loaded_skip_current:REAL;
END_VAR
VAR_OUTPUT
	Auto_ref:REAL;
	Starting_torque:REAL;
	Manual:BOOL;
	Auto:BOOL;
	Auto_go:BOOL;
	Auto_fwd:BOOL;
	Auto_rev:BOOL;
	Trail_brakes:BOOL;
	Fwd_incomplete:BOOL;
	Rev_incomplete:BOOL;
	Left_tip_zone:BOOL;
	Right_tip_zone:BOOL;
	Left_box_zone:BOOL;
	Right_box_zone:BOOL;
	Ready_to_load_rock:BOOL;
	Left_bank_zone:BOOL;
	Right_bank_zone:BOOL;
	ct_Skip_still_full:BOOL;
	ct_Auto_requirements:BOOL;
END_VAR
VAR_IN_OUT
	HMI_data:dut_Auto_rock;
	Levels:ARRAY[*] OF REAL;
END_VAR
VAR
	Auto_requirements_fault:BOOL;
	Rock_cycle_bypass_hmi:BOOL;
	Window_0: FB_Window;
	Window_1: FB_Window;
	R_TRIG_0: R_TRIG;
	R_TRIG_1: R_TRIG;
	TOF_0: TOF;
	F_TRIG_0: F_TRIG;
	BIT_TO_WORD_V0_0: FB_BIT_TO_WORD_V0;
	WORD_TO_BIT_V0_0: FB_WORD_TO_BIT_V0;
END_VAR

M_Zones();
M_Auto_mode();
M_Despatch();
M_Trail_brakes();
M_Auto_trips();
M_HMI_data();

METHOD M_Auto_mode
VAR_INPUT
END_VAR
VAR_INST // added by the converter: edge detectors and wires of the graphical bodies
    _w1, _w2 : BOOL;
    _w3 : ANY;
END_VAR
Auto := (_w1 OR Auto) AND Mode.Auto_switch AND Safety_interlock AND NOT Rock_cycle_bypass_hmi AND Clutch.Rh_in AND Clutch.Lh_in AND Mode.Rock AND _w2 AND Power_leverNeutral AND NOT Brakes.Lever_on AND Brakes.Lever_fully_off AND NOT Brakes.Lh_dump AND NOT Brakes.Rh_dump;
_w2 := Left_tip_zone AND Right_box_zone OR Auto OR Right_tip_zone AND Left_box_zone;
Mode.Auto := _w3;
// Requirements for automatic mode
_w1 := Brakes.Lh_on AND Brakes.Rh_on;
_w3 := Auto;
END_METHOD

METHOD M_Auto_trips
VAR_INPUT
END_VAR
VAR_INST // added by the converter: edge detectors and wires of the graphical bodies
    _w1, _w2, _w3, _w4 : BOOL;
    _w5 : ANY;
END_VAR
ct_skip_still_full := _w1;
_w3 := Fwd_incomplete AND Power_leverReverse OR _w2;
// Trip if the winder moves in the wrong direction in automatic mode
_w2 := Rev_incomplete AND Power_leverForward;
_w1 := _w4 OR _w3 AND NOT Mode.Auto_switch AND NOT Rock_cycle_bypass_hmi;
_w5 := F_TRIG_0.Q AND Mode.Auto_switch;
// Trip if the winder falls out of auto with auto still selected
F_TRIG_0(CLK := Auto); // F_TRIG
ct_Auto_requirements := _w5;
// If a wind was not completed in auto, it must be completed in manual or bypassed in manual to go the other direction
_w4 := (Fwd_incomplete OR Rev_incomplete) AND Mode.Auto_switch AND NOT Auto_go;
END_METHOD

METHOD M_Despatch
VAR_INPUT
END_VAR
VAR_INST // added by the converter: edge detectors and wires of the graphical bodies
    _w1, _w2, _w3, _w4, _w5, _w6, _w7, _w8, _w11, _w12, _w13 : BOOL;
    _w9, _w10 : REAL;
END_VAR
Auto_fwd := _w1;
_w2 := Lh_depth > (Levels[0] + Left_brakes_on_dist);
_w4 := _w3 OR Auto_fwd;
Fwd_incomplete := _w5;
_w6 := Lh_depth > Rock_cycle_unlatch_dist;
_w3 := Right_tip_zone AND Left_box_zone AND Brakes.Lh_on AND Brakes.Rh_on AND Underground_despatch AND _w7;
// Forward cycle
R_TRIG_0(CLK := Underground_despatch); // R_TRIG
_w7 := R_TRIG_0.Q OR Auto_fwd;
Auto_go := _w8;
Starting_torque := _w9;
_w1 := _w4 AND Auto AND NOT Auto_rev AND NOT Rev_incomplete AND _w2;
// Starting current required for fully loaded skip
_w10 := SEL(Auto_fwd, 0, Loaded_skip_current);
// Speed reference in automatic as a percent x100
Auto_ref := SEL(Auto_rev, 32767, -32767);
Auto_fwd := (Left_tip_zone AND Right_box_zone AND Brakes.Lh_on AND Brakes.Rh_on AND Underground_despatch AND _w11 OR Auto_rev) AND Auto AND NOT Auto_rev AND NOT Fwd_incomplete AND _w12;
// Reverse cycle
R_TRIG_1(CLK := Underground_despatch); // R_TRIG
_w11 := R_TRIG_1.Q OR Auto_rev;
_w12 := Rh_depth > (Levels[0] + Right_brakes_on_dist);
// Forward and reverse incomplete cycles
_w5 := (Auto_fwd OR Fwd_incomplete) AND NOT Rev_incomplete AND _w6;
Rev_incomplete := (Auto_rev OR Rev_incomplete) AND NOT Fwd_incomplete AND _w13;
_w13 := Rh_depth > Rock_cycle_unlatch_dist;
// Auto_go bit
_w8 := Auto_fwd OR Auto_rev;
_w9 := SEL(Auto_rev, _w10, Loaded_skip_current);
END_METHOD

METHOD M_HMI_data
VAR_INPUT
END_VAR
HMI_data.Status := BIT_TO_WORD_V0_0.Word_out;
// Pack data for HMI
BIT_TO_WORD_V0_0(
    bit0 := Ready_to_load_rock,
    bit1 := Left_tip_zone,
    bit2 := Left_box_zone,
    bit3 := Right_tip_zone,
    bit4 := Right_box_zone,
    bit5 := Fwd_incomplete,
    bit6 := Rev_incomplete,
    bit7 := Auto_fwd,
    bit8 := Auto_rev,
    bit9 := Underground_despatch); // FB_BIT_TO_WORD_V0
// Data from HMI
WORD_TO_BIT_V0_0(Word_in := HMI_data.Command); // FB_WORD_TO_BIT_V0
Rock_cycle_bypass_hmi := WORD_TO_BIT_V0_0.bit0;
END_METHOD

METHOD M_Trail_brakes
VAR_INPUT
END_VAR
VAR_INST // added by the converter: edge detectors and wires of the graphical bodies
    _w1, _w3 : BOOL;
    _w2 : ANY;
END_VAR
Trail_brakes := TOF_0.Q;
_w1 := Rh_depth < (Levels[0] + 2000) AND Auto_rev;
TOF_0(IN := _w2, PT := Auto_go); // TOF
_w2 := _w3 AND Auto_go;
_w3 := Lh_depth < (Levels[0] + 2000) AND Auto_fwd OR _w1;
END_METHOD

METHOD M_Zones
VAR_INPUT
END_VAR
Right_tip_zone := Window_0.In_window;
Window_1(Minimum := Levels[31] - Box_zone_up, X := Lh_depth, Maximum := Levels[31] + Box_zone_down); // FB_Window
Window_0(Minimum := Levels[0] - Tip_zone_up, X := Lh_depth, Maximum := Levels[0] + Tip_zone_down); // FB_Window
Window_1(Minimum := Levels[31] - Box_zone_up, X := Rh_depth, Maximum := Levels[31] + Box_zone_down); // FB_Window
Left_box_zone := Window_1.In_window;
Window_0(Minimum := Levels[0] - Tip_zone_up, X := Rh_depth, Maximum := Levels[0] + Tip_zone_down); // FB_Window
Left_tip_zone := Window_0.In_window;
Right_box_zone := Window_1.In_window;
END_METHOD

END_FUNCTION_BLOCK

// ---- POUs/FBs/FB_Window.TcPOU
FUNCTION_BLOCK FB_Window
VAR_INPUT
	Minimum:REAL;
	X:REAL;
	Maximum:REAL;
END_VAR
VAR_OUTPUT
	In_window:BOOL;
END_VAR
VAR
END_VAR

M_Window();

METHOD M_Window
VAR_INPUT
END_VAR
In_window := X >= Minimum AND X <= Maximum;
END_METHOD

END_FUNCTION_BLOCK

// ---- POUs/FBs/FB_Backout.TcPOU
FUNCTION_BLOCK FB_Backout
VAR_INPUT
	Backout_switch:BOOL;
	Reset:BOOL;
	Left_overwind:BOOL;
	Left_underwind:BOOL;
	Right_overwind:BOOL;
	Right_underwind:BOOL;
	Brake_lever_on:BOOL;
	Lever_neutral:BOOL;
	Fwd:BOOL;
	Rev:BOOL;
	Forward_backout_relay_fb:BOOL;
	Reverse_backout_relay_fb:BOOL;
END_VAR
VAR_OUTPUT
	Forward_backout_relay:BOOL;
	Reverse_backout_relay:BOOL;
	Forward_xcheck_fault:BOOL;
	Reverse_xcheck_fault:BOOL;
END_VAR
VAR
	Bor_set1:BOOL;
	Bor_set2:BOOL;
	Bor_set3:BOOL;
	Bor_set4:BOOL;
	Bor_rst1:BOOL;
	Bor_rst2:BOOL;
	Bor_rst3:BOOL;
	Bor_rst4:BOOL;
	Bor_rst5:BOOL;
	RS_0: RS;
	TON_0: TON;
	F_TRIG_0: F_TRIG;
END_VAR

M_Backout_main();

METHOD M_Backout_main
VAR_INPUT
END_VAR
VAR_INST // added by the converter: edge detectors and wires of the graphical bodies
    _w1, _w4, _w5, _w7 : BOOL;
    _w2, _w3, _w6 : ANY;
END_VAR
Bor_set1 := _w1;
RS_0(SET := _w2, RESET1 := _w3); // RS
// BOR Relay Activation and Deactivation
_w2 := Bor_set1 OR Bor_set2;
// OW and UW wrong direction detection
Bor_set2 := NOT Right_underwind AND Reset;
Bor_set3 := NOT Right_overwind AND Reset;
Reverse_backout_relay := RS_0.Q1;
// When in either OW or UW on either side, set BOR when Reset PB is pushed.
// The OW and UW signals Fall to Zero when active.
_w1 := NOT Left_overwind AND Reset;
_w3 := Bor_rst1 OR Bor_rst2 OR Bor_rst5 OR Left_overwind AND Right_underwind OR NOT Backout_switch;
Bor_rst2 := NOT Left_overwind AND Fwd;
_w4 := Bor_set3 OR Bor_set4;
Forward_xcheck_fault := TON_0.Q;
_w5 := NOT Left_underwind AND Reset;
TON_0(IN := Reverse_backout_relay XOR Reverse_backout_relay_fb, PT := t#500ms); // TON
RS_0(SET := _w4, RESET1 := _w6); // RS
Bor_set4 := _w5;
Reverse_xcheck_fault := TON_0.Q;
Forward_backout_relay := RS_0.Q1;
_w6 := Bor_rst1 OR Bor_rst4 OR Bor_rst3 OR _w7 OR NOT Backout_switch;
_w7 := Right_overwind AND Left_underwind;
// Backout Relay crosscheck
TON_0(IN := Forward_backout_relay XOR Forward_backout_relay_fb, PT := t#500ms); // TON
// Lever/Brake interlock
F_TRIG_0(CLK := Brake_lever_on); // F_TRIG
Bor_rst1 := Lever_neutral AND F_TRIG_0.Q;
Bor_rst3 := NOT Left_underwind AND Rev;
Bor_rst4 := NOT Right_overwind AND Rev;
Bor_rst5 := NOT Right_underwind AND Fwd;
END_METHOD

END_FUNCTION_BLOCK

// ---- POUs/FBs/FB_Brake.TcPOU
FUNCTION_BLOCK FB_Brake
VAR_INPUT
	Lh_off:BOOL;(*Left brake off signal - usually from left spring nest*)
	Lh_rubbing:BOOL; (*Left brake rubbing signal - usually from left spring nest*)
	Lh_on:BOOL; (*Left brake on signal - usually from left spring nest*)
	Lh_wear:BOOL; (*Left brake wear signal - usually from left spring nest*)
	Rh_off:BOOL; (*Right brake on signal - usually from right spring nest*)
	Rh_rubbing:BOOL; (*Right brake rubbing signal - usually from right spring nest*)
	Rh_on:BOOL; (*Right brake on signal - usually from right spring nest*)
	Rh_wear:BOOL; (*Right brake wear signal - usually from Right spring nest*)
	Lever_on:BOOL; (*Brake lever on limit switch*)
	Lever_off:BOOL; (*Brake lever off - normally from same limit switch as "Lever_on"*)
	Lever_fully_off:BOOL; (*Brake lever fully off limit switch. Necessary for automatic winders.*)
	Lh_test:BOOL; (*Left brake test switch - normally on driver's desk. Often the same switch as Lh_dump.*)
	Rh_test:BOOL; (*Right brake test switch - normally on driver's desk. Often the same switch as Rh_dump.*)
	Lh_dump:BOOL; (*Left brake dump switch - normally on driver's desk. Often the same switch as Lh_test.*)
	Rh_dump:BOOL; (*Right brake dump switch - normally on driver's desk. Often the same switch as Rh_test.*)
	Maintenance_switch:BOOL; (*Brake maintenance switch (can be on driver's desk or in control panels).*)
	Trail_brakes:BOOL; (*Trail brake control signal. Used to disable Lh_not_fully_off and Rh_not_fully_off trips.*)
	Lh_speed:INT; (*Left drum speed (normally in mm/s)*)
	Rh_speed:INT; (*Right drum speed (normally in mm/s)*)
	Movement_detect:BOOL; (*Drum movement detected (on either of the two drums in a double-drum winder)*)
	On_time:TIME; (*Maximum time allowed for brakes to apply.*)
	Off_time:TIME; (*Maximum time allowed for brakes to lift.*)
	Rubbing_speed:INT; (*Speed above which the brakes must be above the rubbing position*)
	Rubbing_time:TIME; (*Time before brake rubbing trips trigger *)
END_VAR
VAR_OUTPUT
	Maintenance:BOOL; (*The winder is in brake maintenance mode*)
	Proved_on:BOOL; (*The brake lever (if in manual mode) and both brakes are on*)
	Proved_on_500ms:BOOL; (*The brakes have been proved on for 500ms*)
	cs_Lh_off_before_rubbing:BOOL; (*The Lh_off switch has closed but the Lh_rubbing switch has not yet closed*)
	cs_Lh_on_and_rubbing:BOOL; (*The Lh_on switch has closed but the Lh_rubbing switch is still closed*)
	cs_Lh_wear_before_on:BOOL; (*The Lh_on switch has closed but the Lh_rubbing switch is still closed*)
	cs_Lh_on_and_off:BOOL; (*The Lh_on and Lh_off switches are simultaneously closed*)
	cs_Rh_off_before_rubbing:BOOL; (*The Rh_off switch has closed but the Rh_rubbing switch has not yet closed*)
	cs_Rh_on_and_rubbing:BOOL; (*The Rh_on switch has closed but the Rh_rubbing switch is still closed*)
	cs_Rh_wear_before_on:BOOL; (*The Rh_on switch has closed but the Rh_rubbing switch is still closed*)
	cs_Rh_on_and_off:BOOL; (*The Rh_on and Rh_off switches are simultaneously closed*)
	cs_Lever_off_and_on:BOOL; (*The brake lever on and off switches are simultaneously closed*)
	cs_Lever_fully_off_and_on:BOOL; (*The brake lever on and fully off switches are simultaneously closed*)
	cs_Lh_not_fully_off:BOOL; (*The brake lever has been off for longer than the brake lift time but the Lh_off switch is not closed. Trail_brakes disables this fault.*)
	cs_Rh_not_fully_off:BOOL; (*The brake lever has been off for longer than the brake lift time but the Rh_off switch is not closed. Trail_brakes disables this fault.*)
	tr_Lh_not_on:BOOL; (*The brake lever has been on for longer than the brake application time but the Lh_on switch is not closed.*)
	tr_Rh_not_on:BOOL; (*The brake lever has been on for longer than the brake application time but the Rh_on switch is not closed.*)
	tr_Lh_rubbing_trip:BOOL; (*Lh_rubbing active above the rubbing trip speed*)
	tr_Rh_rubbing_trip:BOOL; (*Rh_rubbing active above the rubbing trip speed*)
	tr_No_brake_on_in_maint:BOOL; (*The power lever was moved from the neutral position in brake maintenance mode*)
	tr_Movement_in_maint:BOOL; (*Movement has been detected in brake maintenance mode*)
	tr_Maint_switch_on:BOOL; (*The brake maintenance switch is on but a brake is not dumped*)
	hmi_Status:ARRAY[1..2] OF WORD; (*Status bits for HMI*)
END_VAR
VAR
	TON_0: TON;
	Maintenance_req: BOOL;
	RS_0: RS;
	TON_1: TON;
	TON_2: TON;
	TON_3: TON;
	TON_4: TON;
	TON_5: TON;
	TON_6: TON;
	TON_7: TON;
	TON_8: TON;
	TON_9: TON;
	TON_10: TON;
	TON_11: TON;
	TON_12: TON;
	TON_13: TON;
	TON_14: TON;
	TON_15: TON;
	TON_16: TON;
	TON_17: TON;
	BIT_TO_WORD_V0_0: FB_BIT_TO_WORD_V0;
	BIT_TO_WORD_V0_1: FB_BIT_TO_WORD_V0;
END_VAR

M_Brake_data();
M_Brake_faults();

METHOD M_Brake_data
VAR_INPUT
END_VAR
VAR
END_VAR
VAR_INST // added by the converter: edge detectors and wires of the graphical bodies
    _w1 : BOOL;
END_VAR
BIT_TO_WORD_V0_0(
    bit0 := Lh_off,
    bit1 := Lh_rubbing,
    bit2 := Lh_on,
    bit3 := Lh_wear,
    bit4 := Rh_off,
    bit5 := Rh_rubbing,
    bit6 := Rh_on,
    bit7 := Rh_wear,
    bit8 := Lever_on,
    bit9 := Lever_off,
    bit10 := Lever_fully_off,
    bit11 := Lh_test,
    bit12 := Rh_test,
    bit13 := Lh_dump,
    bit14 := Rh_dump,
    bit15 := Maintenance_switch); // FB_BIT_TO_WORD_V0
// Brake data section
// Pack data in Brakes structure
Brakes.Lh_on := Lh_on;
Brakes.Lh_rubbing := Lh_rubbing;
Brakes.Lever_on := Lever_on;
hmi_Status[1] := BIT_TO_WORD_V0_0.Word_out;
Brakes.Lh_off := Lh_off;
Brakes.Lh_wear := Lh_wear;
Brakes.Lever_off := Lever_off;
Brakes.Rh_on := Rh_on;
Brakes.Rh_rubbing := Rh_rubbing;
Brakes.Lever_fully_off := Lever_fully_off;
Brakes.Rh_off := Rh_off;
Brakes.Rh_wear := Rh_wear;
Brakes.Lh_dump := Lh_dump;
Brakes.Rh_dump := Rh_dump;
Brakes.Lh_test := Lh_test AND Clutch.Lh_in;
Brakes.Rh_test := Rh_test AND Clutch.Rh_in;
hmi_Status[2] := BIT_TO_WORD_V0_1.Word_out;
// Brake proving
Brakes.Proved_on := Proved_on;
Proved_on := (Lever_on OR Mode.Auto) AND Lh_on AND Rh_on;
Brakes.Proved_on_500ms := Proved_on_500ms;
TON_0(IN := Proved_on, PT := t#500ms); // TON
Proved_on_500ms := TON_0.Q;
// Brake Maintenance
_w1 := Maintenance_switch;
BIT_TO_WORD_V0_1(bit0 := Proved_on, bit1 := Proved_on_500ms, bit2 := Maintenance); // FB_BIT_TO_WORD_V0
Brakes.Maintenance_switch := _w1;
Maintenance_req := (Lh_dump OR Rh_dump) AND Maintenance_switch;
RS_0(SET := Maintenance_req AND Brakes.Proved_on_500ms, RESET1 := Maintenance_req); // RS
Maintenance := RS_0.Q1;
Brakes.Maintenance_mode := Maintenance;
END_METHOD

METHOD M_Brake_faults
VAR_INPUT
END_VAR
VAR_INST // added by the converter: edge detectors and wires of the graphical bodies
    _w1, _w2, _w4 : BOOL;
    _w3 : ANY;
END_VAR
